(* Logix 5000 project; controller Reto1_SeparatingEstation2 Emulate 5570 rev 30.12; software revision 30.00 *)

TASK MainTask (continuous, watchdog 500 ms) : MainProgram

MODULES
   Local : Emulate 5570 (ICP 2, rev 30.12)
      I_O : vendor 1 type 0 code 15 (ICP 3, rev 1.1, Output RPI 150 ms)
END_MODULES

VAR_GLOBAL   (* controller tags *)
   Banda1 : BOOL;
   Banda1b : BOOL := 1;
   Banda2 : BOOL := 1;
   Banda2b : BOOL := 1;
   BanderaSenA : BOOL;
   ParadaA : BOOL;
   ParadaUPA : BOOL;
   PusherAzul : BOOL;
   Retomar : BOOL;
   senAzul : BOOL;
   SensorAzul : BOOL;
   SensorPaso2 : BOOL;
   SensorVerde : BOOL;
   Start : BOOL;
   Starter : BOOL;   // inicializar pusher
   Stop : BOOL := 1;
   Stop_emergencia : BOOL := 1;
   TimerP : TIMER := (PRE := 2000);
   TimerR : TIMER := (PRE := 2000);
END_VAR

PROGRAM MainProgram   (* main routine MainRoutine *)
VAR
   Counter1 : COUNTER := (PRE := 5);
END_VAR

ROUTINE Ambas   (* ladder *)
END_ROUTINE

ROUTINE Azul   (* ladder *)
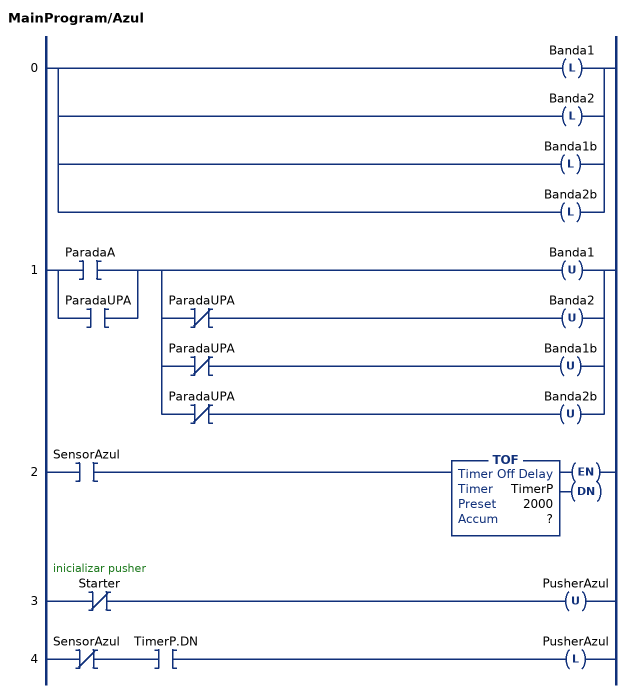
   0: [OTL(Banda1) ,OTL(Banda2) ,OTL(Banda1b) ,OTL(Banda2b) ];
   1: [XIC(ParadaA) ,XIC(ParadaUPA) ][OTU(Banda1) ,XIO(ParadaUPA) OTU(Banda2) ,XIO(ParadaUPA) OTU(Banda1b) ,XIO(ParadaUPA) OTU(Banda2b) ];
   2: XIC(SensorAzul)TOF(TimerP,?,?);
   3: XIO(Starter)OTU(PusherAzul);
   4: XIO(SensorAzul)XIC(TimerP.DN)OTL(PusherAzul);
END_ROUTINE

ROUTINE MainRoutine   (* ladder *)
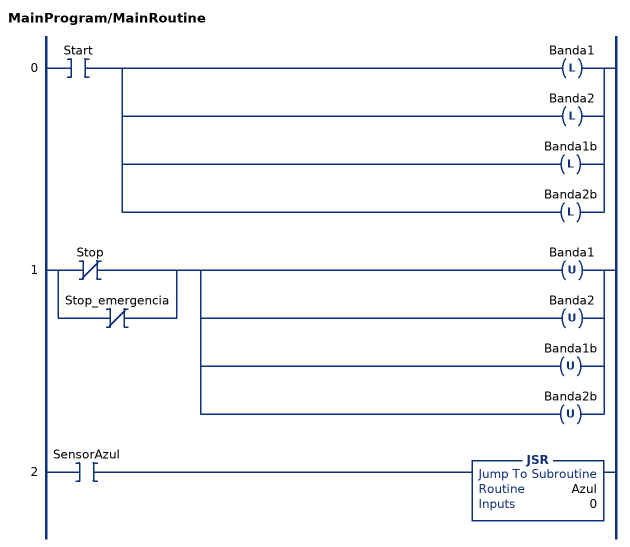
   0: XIC(Start)[OTL(Banda1) ,OTL(Banda2) ,OTL(Banda1b) ,OTL(Banda2b) ];
   1: [XIO(Stop) ,XIO(Stop_emergencia) ][OTU(Banda1) ,OTU(Banda2) ,OTU(Banda1b) ,OTU(Banda2b) ];
   2: XIC(SensorAzul)JSR(Azul,0);
END_ROUTINE
END_PROGRAM
